{attribute 'linkalways'} 
{attribute 'no_explicit_call' := 'This FB is a CLASS and must be accessed using methods or properties'}
{attribute 'enable_dynamic_creation'}
FUNCTION_BLOCK _ETcVnPaddingMode EXTENDS EnumDatatypeBase
VAR
	localData : ETcVnPaddingMode;
	activeData : REFERENCE TO ETcVnPaddingMode;
	enumBaseDatatype : _DINT(localData);
END_VAR

METHOD PRIVATE AddLocalEnumeration
VAR_INPUT
	Enumeration : T_MAXSTRING;
	Value : ETcVnPaddingMode;
END_VAR
AddEnumeration(Enumeration, Value);
END_METHOD

PROPERTY PUBLIC Address : PVOID
GET
Address := ADR(activeData);
END_GET
END_PROPERTY

METHOD PUBLIC ClearReference
VAR_INPUT
END_VAR
activeData REF= localData;
SetBaseDatatypeReference();
END_METHOD

METHOD PUBLIC Clone : I_Datatype
VAR
    pClone : POINTER TO _ETcVnPaddingMode;
END_VAR
pClone := __NEW(_ETcVnPaddingMode(InitialValue := Value));
Clone := pClone^;
END_METHOD

METHOD FB_init : BOOL
VAR_INPUT
	bInitRetains : BOOL; // if TRUE, the retain variables are initialized (warm start / cold start)
	bInCopyCode : BOOL;  // if TRUE, the instance afterwards gets moved into the copy code (online change)
	InitialValue : ETcVnPaddingMode;
END_VAR
localData := InitialValue;
AddBaseDatatype(enumBaseDatatype);
ClearReference();

AddLocalEnumeration('TCVN_PM_NONE', ETcVnPaddingMode.TCVN_PM_NONE);
AddLocalEnumeration('TCVN_PM_CROP_CENTER', ETcVnPaddingMode.TCVN_PM_CROP_CENTER);
AddLocalEnumeration('TCVN_PM_LETTERBOX', ETcVnPaddingMode.TCVN_PM_LETTERBOX);
END_METHOD

PROPERTY PUBLIC Identifier : T_MAXSTRING
GET
Identifier := 'ETcVnPaddingMode';
END_GET
END_PROPERTY

METHOD IsEnumeratorValueEqual : BOOL
VAR_INPUT
	Enumerator : I_KeyValueForwardEnumerator;
END_VAR
VAR
	storedValue : ETcVnPaddingMode;
END_VAR
IF NOT Enumerator.TryGet(storedValue) THEN
	RETURN;
END_IF

IsEnumeratorValueEqual := storedValue = activeData;
END_METHOD

METHOD PUBLIC MakeReferenceTo
VAR_INPUT
	ReferenceTarget : REFERENCE TO ETcVnPaddingMode;
END_VAR
activeData REF= ReferenceTarget;
SetBaseDatatypeReference();
END_METHOD

METHOD PROTECTED SetBaseDatatypeReference
VAR_INPUT
END_VAR
enumBaseDatatype.MakeReferenceTo(activeData);
END_METHOD

PROPERTY PUBLIC Size : UDINT
GET
Size := SIZEOF(activeData);
END_GET
END_PROPERTY

METHOD TryMakeReferenceTo : BOOL
VAR_INPUT
	Target : I_Datatype;
END_VAR
VAR
	targetAsEnum : I_EnumDatatype;
	pTargetData : POINTER TO ETcVnPaddingMode;
END_VAR
IF NOT Target.TryResolveAsEnumDatatype(targetAsEnum) THEN
	RETURN;
END_IF

IF targetAsEnum.Identifier <> Identifier THEN
	RETURN;
END_IF

pTargetData := Target.Address;
activeData REF= pTargetData^;
SetBaseDatatypeReference();
TryMakeReferenceTo := TRUE;
END_METHOD

PROPERTY PUBLIC Value : ETcVnPaddingMode
GET
Value := activeData;
END_GET
SET
activeData := Value;
END_SET
END_PROPERTY

END_FUNCTION_BLOCK

(* stored: Version 1.1.0.1, ProductVersion 3.1.4024.13
   POU _ETcVnPaddingMode: Id {bbe1ad36-8b57-02bc-1621-e2b0acd71e20}, SpecialFunc None
   Folder Core: Id {2ed99e2a-91da-000f-24e9-073793b5fe88}
   Folder Protected: Id {cc33437f-1d56-0606-17f3-a94731d6d370}
   Folder Customize: Id {27ab5f09-2d67-0c47-2256-a0b528669063}
   Folder Constructor: Id {af6f6a35-0601-0b9e-3974-c3a6e31844d6}
   Folder Private: Id {c6df4e62-1d61-0986-0b5a-319dc79c6aec}
   Folder Protected: Id {334c2d1d-29e0-02e2-3643-feb7b45dd40c}
   Method AddLocalEnumeration: Id {634c9caa-4e8d-083d-2b40-c030df59ea1c}
   Property Address: Id {8078aad7-f0c5-057f-018a-9cb870b16fb8}
   Get Get: Id {b01e1835-da28-02e9-2d95-e7ae04ed30de}
   Method ClearReference: Id {6813acf9-6457-0a19-2f67-5c03d50086f3}
   Method Clone: Id {4fa31f1e-601a-0f57-243d-9b3f6fc53ea0}
   Method FB_init: Id {3ed9770d-9286-0795-0cce-1ae8a7929af7}
   Property Identifier: Id {6366a64e-0e08-0a97-2e7e-7d3db35a073a}
   Get Get: Id {dbfadd98-6e16-040f-1614-64bee2042a1c}
   Method IsEnumeratorValueEqual: Id {332d08c5-555e-0c39-3040-96311f7b944c}
   Method MakeReferenceTo: Id {defff4a0-2b24-0342-35f8-75c5484c69cb}
   Method SetBaseDatatypeReference: Id {4d99bf1a-ba32-0ef8-0d9f-88ddc4d2451f}
   Property Size: Id {81fab8b6-79a8-0742-1803-f014509f95cb}
   Get Get: Id {93183db2-33b5-046a-0722-973cae55d6ce}
   Method TryMakeReferenceTo: Id {846ad209-dfc4-0303-30ac-3c483e6518eb}
   Property Value: Id {3c8a1d12-8adb-065c-2b05-8456703512d1}
   Get Get: Id {e7be3f0f-7fa0-0a22-2851-c6f307fc95e3}
   Set Set: Id {04771c5a-c636-0a02-131b-2ebe3333d8bf} *)
